// TIA Portal V19 export
DATA_BLOCK "DB_POS"   // DB51
{ S7_Optimized_Access := 'FALSE' }
AUTHOR : MS
// stored: AutoNumber false
   VAR RETAIN
      ANZAHL : Int := 58;   // Anzahl der Positionen
      Offset : Int := 50;   // * Beginn der Datenstruktur
      LENG : Int := 100;   // * Länge einer Position in Byte
      akt_POS : Int := 13;   // Position in Bearbeitung
      resW : Int := 0;
      resDW1 : DWord := 16#0000_0000;
      RESDW2 : DWord := 16#0000_0000;
      RESDW3 : DWord := 16#0000_0000;
      RESDW4 : DWord := 16#0000_0000;
      RESDW5 : DWord := 16#0000_0000;
      RESDW6 : DWord := 16#0000_0000;
      RESDW7 : DWord := 16#0000_0000;
      RESDW8 : DWord := 16#0000_0000;
      RESDW9 : DWord := 16#0000_0000;
      RESDW10 : DWord := 16#0000_0000;
      POS : Array[0..30] of Struct   // * Feldlänge anpassen
         Typ : Byte;   // Badtyp 0=Anlagenpos normal, 1-3=Be-Entladestand, 5=Speicher ,10=QT-Pos, 255 Dum
         SubTyp : Byte;   // Untertyp der Position 5=ExpoVorruf ignorieren bei 2xEinsetzen, 1=Sperre bei Alt
         Prio_Pos : Byte;   // Priorität des Bades (höchste Priorität==0
         SchiebePos : Byte;   // Position auf die FW geschoben wird, wenn er ohne Befehl hier steht
         Reihe : Byte;   // Reihe auf der sich die Position befindet
         FW_Nr : Byte;   // FW_Nr des FW, der über dieser Pos ist
         Optipos : Bool;   // WT wird in die Optimierungsrechnung einbezogen
         berechnet : Bool;   // WT wurde von der Optimierung berechnet
         Quelle : Bool;   // Position ist als Quelle reserviert
         Ziel : Bool;   // Position ist als Ziel reserviert
         FW_kommt : Bool;   // FW will dieses Bad überfahren
         FW_in_POS : Bool;   // Fahrwagen über Bad positioniert
         FW_Hebt : Bool;   // Fahrwagen hebt aus
         FW_Senkt : Bool;   // Fahrwagen setzt ein
         Sperre_in : Bool;   // Bad Einfahrsperre
         Sperre_FW : Bool;   // Bad Überfahrsperre
         Sperre_out : Bool;   // Bad Ausfahrsperre
         IN_OUT_nen : Bool;   // Einsetzen bzw. Ausheben nicht möglich, da Warenbewegung oder Deckel zu usw.
         lngsm_IN : Bool;   // langsames Einsetzen erforderlich-abhängig von immer_schnell
         lngsm_OUT : Bool;   // langsames Ausheben erforderlich-abhängig von immer_schnell
         immer_schnell : Bool;   // trockene Position (keine ATZ, schneller Hub erlaubt)
         QT_reserviert : Bool;   // Position ist durch QT reserviert
         KS_erlaubt : Bool;   // Pos darf mit KS befülltwerden
         LS_erlaubt : Bool;   // Pos darf mit LS befüllt werden
         GO_erlaubt : Bool;   // Pos darf mit GO befüllt werden
         Belegt_KS : Bool;   // Belegt mit KS
         Belegt_LS : Bool;   // Belegt mit LS
         Belegt_GO : Bool;   // Belegtmit GO
         Spr_Off : Bool;   // Oberhalb Z nicht spritzen
         Opt_Abgelehnt : Bool;   // Einfahrt durch Opti abgelehnt
         notFG_out : Bool;   // Position darf nicht geräumt werden (Merkersystem)
         notFG_in : Bool;   // Position darf nicht befüllt werden (Merkersystem)
         Anmeldung : Bool;   // bevorzugte Behandlung anmelden
         fPosfree : Bool;   // Folgeposition muß frei sein
         QT_Sperre : Bool;   // Position ist durch QT gesperrt FW darf Pos nicht bedienen
         Vorsperre : Bool;   // Einfahrsperre anmelden
         QT_FW_Ruf : Bool;   // QT wird auf dieser Position von einem FW benötigt
         QT_ext_Ruf : Bool;   // QT wird auf dieser Position von einem externen Gerät benötigt
         Bef_ende : Bool;   // in diesem Bad muß der Befehlsindex geschaltet werden
         DoppelTauch : Bool;   // Doppeltauchen angefordert
         ignor_Exp : Bool;   // Expozeit ignorieren (Transport)
         ignor_ESp : Bool;   // ignoriere Einfahrsperre (notFG_in)
         ignor_fPosFree : Bool;   // ignoriere fPosFree (z.B. für Freigabe Pos kurz vor Expoende)
         UebergabePos : Bool;   // Übergabe von Wts möglich
         Portable : Bool;   // Im Vorruf und transportierbar
         Checked : Bool;   // Position im ersten Check (FB9) geprüft
         Detailtyp : Byte;   // 0=egal, 11=KS. 12=LS, 20=GO (alleshex)
         BereichsTakte : Byte;   // 0=kein laden, ansonsten auf WTDB.DBB54
         Stand_Nr : Byte;   // Verweis auf Stand Nr
         Absetzhoehe : DInt;   // Absetzhöhe in Inkrementen
         LZ_Nr1 : Byte;   // Verweis auf Ladungszähler Nr1
         LZ_Nr2 : Byte;   // Verweis auf Ladungszähler Nr2
         ZG_1 : Byte;   // Reserve für weitere Verweise
         ZG_2 : Byte;   // Reserve für weitere Verweise
         IncPos : DInt;   // Position des Bades in der Anlage
         IncAbstand_vor : Int;   // min. Abstand zum Bad bei Überfahrsperre
         IncAbstand_rck : Int;   // min. Abstand zum Bad bei Überfahrsperre
         WT_Nr_lang : DInt;   // Warenträger-Nr.
         WT_Stangen_Nr : Byte;   // Stangen-Nr
         WT_DB : Byte;   // DB_Nr Warenstange
         next_WT : Byte;   // WT der sich für diese Pos anmeldet
         Prio : Bool;
         INA : Bool;
         INE : Bool;
         OUTA : Bool;
         OUTE : Bool;
         SpProg : Bool;
         ResAmTW : Bool;
         ResAmQT : Bool;
         Trommel : Bool;   // Kontrolle aktiviert
         Leer_WT : Bool;   // Leerwarenträger HFs aus
         Warnung : Bool;   // in Position wurde eine Warnmeldung ausgelöst
         Alarm : Bool;   // in Position wurde eine Alarmmeldung ausgelöst
         WT_neu : Bool;   // WT wurde vom LZ noch nicht berücksichtigt
         lngsm_Hub : Bool;   // langsam Heben als WT-Parameter
         B_Takte_Null : Bool;   // Bereichstakte sind Null
         enable_reload : Bool;   // laden der Altwerte innerhalb einer Gruppe erlaubt
         WT_Typ : Byte;   // Art des Warenträgers (z.Bsp. bei fester Zuordnung Ware-WT)
         WT_Befx : Int;   // WT Befehlsindex
         Soll_Takte : Int;   // VERWEILTAKTE
         Soll_Expozeit : DInt;   // Sollwert Expositionszeit
         ExpoToleranz : DInt;   // Toleranzwert für Expozeit
         KF_A : Real;   // Korrekturfaktor WT_Auslastung 0..100%-->0..1, Gesamtoberfläche
         KF_Expo : Real;   // Korrekturfaktor Expozeit
         Korr_Restzeit : DInt;   // korregierte Restzeit bis zur Abholung WT
         SonderPos_Offset : DInt;   // Offset für Positionierung außermittig (Höhenwechsel,Blende usw.)
         Restvorsperre : Int;   // Resttakte bis Vorsperre
         Resttakte : Int;   // Taktzähler
         Restzeit : DInt;   // verbleibende Expositionszeit
         Verweilzeit : DInt;   // Verweilzeit
         T_Vorruf : Int;   // Vorrufzeit lößt Vorruf n Sekunden vor Ablauf der Expozeit aus
         T_Pend : Int;   // Auspendelzeit 0..999s
         T_ATZ : Int;   // Abtropfzeit 0..999s
         T_Vorsperre : Int;   // Takte bis Vorsperre zu Sperre wird
         WaitTime : DInt;   // Zeit der Expounterbrechung
         Res_Real : Real;
         belegt : Bool;   // Bad belegt
         Bearbeitung : Bool;   // Badbehandlung läuft
         Vorruf : Bool;   // Bad FW-Vorruf
         fertig : Bool;   // Bad fertig
         AL_Expo : Bool;   // Expotoleranz um 30s überschritten
         Dkl_auf_Pos : Bool;
         Expo_Off : Bool;   // Expozeit unterbrochen (GR-Absenkung)
         yALEX : Bool;   // Alarm Expo auslösen
         US_on_Q : Bool;   // Ultraschall 7s einschalten, wenn Quelle
         AlExp : Bool;   // Alarm Expotoleranz war ein
         MD_Alex : Bool;   // Meldung Expoalarm wurde abgesetzt
         MD_res : Bool;   // Meldung Gleichrichterfehler
         MD_res_1 : Bool;   // Meldung Temperaturreglerfehler
         QT_in_Pos : Bool;   // QT in Position
         res27 : Bool;
         PendHub : Bool;   // Pendelhub aktiv
         Leerzeit : Int;   // Zeit welche Position nicht benutzt
      END_STRUCT;
      RESDW : DWord := 16#0000_0000;
   END_VAR
BEGIN
   POS[0].Typ := 16#00;
   POS[1].Typ := 16#03;
   POS[2..30].Typ := 16#00;
   POS[0..30].SubTyp := 16#00;
   POS[0..30].Prio_Pos := 16#05;
   POS[0..30].SchiebePos := 16#00;
   POS[0..30].Reihe := 16#01;
   POS[0..1].FW_Nr := 16#00;
   POS[2].FW_Nr := 16#01;
   POS[3..10].FW_Nr := 16#00;
   POS[11].FW_Nr := 16#02;
   POS[12..30].FW_Nr := 16#00;
   POS[0..30].Optipos := FALSE;
   POS[0..30].berechnet := FALSE;
   POS[0..30].Quelle := FALSE;
   POS[0..30].Ziel := FALSE;
   POS[0..30].FW_kommt := FALSE;
   POS[0..1].FW_in_POS := FALSE;
   POS[2].FW_in_POS := TRUE;
   POS[3..10].FW_in_POS := FALSE;
   POS[11].FW_in_POS := TRUE;
   POS[12..30].FW_in_POS := FALSE;
   POS[0..30].FW_Hebt := FALSE;
   POS[0..30].FW_Senkt := FALSE;
   POS[0..30].Sperre_in := FALSE;
   POS[0..30].Sperre_FW := FALSE;
   POS[0..30].Sperre_out := FALSE;
   POS[0..30].IN_OUT_nen := FALSE;
   POS[0..30].lngsm_IN := FALSE;
   POS[0..30].lngsm_OUT := FALSE;
   POS[0].immer_schnell := FALSE;
   POS[1..2].immer_schnell := TRUE;
   POS[3..27].immer_schnell := FALSE;
   POS[28].immer_schnell := TRUE;
   POS[29..30].immer_schnell := FALSE;
   POS[0..30].QT_reserviert := FALSE;
   POS[0..30].KS_erlaubt := FALSE;
   POS[0..30].LS_erlaubt := FALSE;
   POS[0..30].GO_erlaubt := FALSE;
   POS[0..30].Belegt_KS := FALSE;
   POS[0..30].Belegt_LS := FALSE;
   POS[0..30].Belegt_GO := FALSE;
   POS[0..30].Spr_Off := FALSE;
   POS[0..30].Opt_Abgelehnt := FALSE;
   POS[0].notFG_out := FALSE;
   POS[1].notFG_out := TRUE;
   POS[2..30].notFG_out := FALSE;
   POS[0].notFG_in := FALSE;
   POS[1].notFG_in := TRUE;
   POS[2..30].notFG_in := FALSE;
   POS[0..30].Anmeldung := FALSE;
   POS[0..30].fPosfree := FALSE;
   POS[0..30].QT_Sperre := FALSE;
   POS[0..30].Vorsperre := FALSE;
   POS[0..30].QT_FW_Ruf := FALSE;
   POS[0..30].QT_ext_Ruf := FALSE;
   POS[0..30].Bef_ende := TRUE;
   POS[0..30].DoppelTauch := FALSE;
   POS[0..30].ignor_Exp := FALSE;
   POS[0..30].ignor_ESp := FALSE;
   POS[0..30].ignor_fPosFree := FALSE;
   POS[0..30].UebergabePos := FALSE;
   POS[0..30].Portable := FALSE;
   POS[0..30].Checked := FALSE;
   POS[0..9].Detailtyp := 16#00;
   POS[10].Detailtyp := 16#16;
   POS[11..12].Detailtyp := 16#00;
   POS[13].Detailtyp := 16#15;
   POS[14].Detailtyp := 16#14;
   POS[15..16].Detailtyp := 16#00;
   POS[17].Detailtyp := 16#13;
   POS[18].Detailtyp := 16#00;
   POS[19].Detailtyp := 16#12;
   POS[20..21].Detailtyp := 16#00;
   POS[22].Detailtyp := 16#11;
   POS[23..30].Detailtyp := 16#00;
   POS[0..30].BereichsTakte := 16#00;
   POS[0].Stand_Nr := 16#00;
   POS[1].Stand_Nr := 16#01;
   POS[2..30].Stand_Nr := 16#00;
   POS[0..30].LZ_Nr1 := 16#00;
   POS[0..30].LZ_Nr2 := 16#00;
   POS[0..30].ZG_1 := 16#00;
   POS[0..30].ZG_2 := 16#00;
   POS[0].IncPos := 12000;
   POS[1].IncPos := 1000;
   POS[2].IncPos := 2000;
   POS[3].IncPos := 3000;
   POS[4].IncPos := 4000;
   POS[5].IncPos := 5000;
   POS[6].IncPos := 6000;
   POS[7].IncPos := 7000;
   POS[8].IncPos := 8000;
   POS[9].IncPos := 9000;
   POS[10].IncPos := 10000;
   POS[11].IncPos := 11000;
   POS[12].IncPos := 12000;
   POS[13].IncPos := 13000;
   POS[14].IncPos := 14000;
   POS[15].IncPos := 15000;
   POS[16].IncPos := 16000;
   POS[17].IncPos := 17000;
   POS[18].IncPos := 18000;
   POS[19].IncPos := 19000;
   POS[20].IncPos := 20000;
   POS[21].IncPos := 21000;
   POS[22].IncPos := 22000;
   POS[23].IncPos := 23000;
   POS[24].IncPos := 24000;
   POS[25].IncPos := 25000;
   POS[26].IncPos := 26000;
   POS[27].IncPos := 27000;
   POS[28].IncPos := 28000;
   POS[29].IncPos := 29000;
   POS[30].IncPos := 30000;
   POS[0].IncAbstand_vor := 0;
   POS[1].IncAbstand_vor := 600;
   POS[2..30].IncAbstand_vor := 0;
   POS[0].IncAbstand_rck := 0;
   POS[1].IncAbstand_rck := 300;
   POS[2..30].IncAbstand_rck := 0;
   POS[0..30].WT_Nr_lang := 0;
   POS[0..30].WT_Stangen_Nr := 16#00;
   POS[0..30].WT_DB := 16#00;
   POS[0..30].next_WT := 16#00;
   POS[0..30].Prio := FALSE;
   POS[0..30].INA := FALSE;
   POS[0..30].INE := FALSE;
   POS[0..30].OUTA := FALSE;
   POS[0..30].OUTE := FALSE;
   POS[0..30].SpProg := FALSE;
   POS[0..30].ResAmTW := FALSE;
   POS[0..30].ResAmQT := FALSE;
   POS[0..30].Trommel := FALSE;
   POS[0..30].Leer_WT := FALSE;
   POS[0..30].Warnung := FALSE;
   POS[0..30].Alarm := FALSE;
   POS[0..30].WT_neu := FALSE;
   POS[0..30].lngsm_Hub := FALSE;
   POS[0..30].B_Takte_Null := FALSE;
   POS[0..3].enable_reload := FALSE;
   POS[4..7].enable_reload := TRUE;
   POS[8..30].enable_reload := FALSE;
   POS[0..30].WT_Typ := 16#00;
   POS[0..30].WT_Befx := 0;
   POS[0..30].Soll_Takte := 0;
   POS[0].Soll_Expozeit := 5;
   POS[1].Soll_Expozeit := 0;
   POS[2].Soll_Expozeit := 360;
   POS[3].Soll_Expozeit := 60;
   POS[4..7].Soll_Expozeit := 1260;
   POS[8..9].Soll_Expozeit := 90;
   POS[10].Soll_Expozeit := 75;
   POS[11..12].Soll_Expozeit := 5;
   POS[13..14].Soll_Expozeit := 75;
   POS[15..16].Soll_Expozeit := 5;
   POS[17].Soll_Expozeit := 75;
   POS[18].Soll_Expozeit := 5;
   POS[19].Soll_Expozeit := 75;
   POS[20].Soll_Expozeit := 5;
   POS[21].Soll_Expozeit := 10;
   POS[22].Soll_Expozeit := 360;
   POS[23..27].Soll_Expozeit := 5;
   POS[28].Soll_Expozeit := 0;
   POS[29..30].Soll_Expozeit := 5;
   POS[0..30].ExpoToleranz := 600;
   POS[0..30].KF_A := 0.0;
   POS[0..30].KF_Expo := 0.0;
   POS[0..30].Korr_Restzeit := 0;
   POS[0..30].SonderPos_Offset := 0;
   POS[0..30].Restvorsperre := 0;
   POS[0..30].Resttakte := 0;
   POS[0..30].Restzeit := 0;
   POS[0..30].Verweilzeit := 0;
   POS[0..30].T_Vorruf := 30;
   POS[0..30].T_Pend := 1;
   POS[0].T_ATZ := 5;
   POS[1..2].T_ATZ := 0;
   POS[3..7].T_ATZ := 10;
   POS[8..9].T_ATZ := 5;
   POS[10].T_ATZ := 10;
   POS[11..12].T_ATZ := 5;
   POS[13..14].T_ATZ := 10;
   POS[15..16].T_ATZ := 5;
   POS[17].T_ATZ := 10;
   POS[18].T_ATZ := 5;
   POS[19].T_ATZ := 10;
   POS[20..21].T_ATZ := 5;
   POS[22].T_ATZ := 10;
   POS[23].T_ATZ := 5;
   POS[24..27].T_ATZ := 2;
   POS[28].T_ATZ := 0;
   POS[29].T_ATZ := 5;
   POS[30].T_ATZ := 2;
   POS[0..30].T_Vorsperre := 0;
   POS[0..30].WaitTime := 0;
   POS[0..30].Res_Real := 0.0;
   POS[0..30].belegt := FALSE;
   POS[0..30].Bearbeitung := FALSE;
   POS[0..30].Vorruf := FALSE;
   POS[0..30].fertig := FALSE;
   POS[0..30].AL_Expo := FALSE;
   POS[0..30].Dkl_auf_Pos := FALSE;
   POS[0..30].Expo_Off := FALSE;
   POS[0..30].yALEX := FALSE;
   POS[0..30].US_on_Q := FALSE;
   POS[0..30].AlExp := FALSE;
   POS[0..30].MD_Alex := FALSE;
   POS[0..30].MD_res := FALSE;
   POS[0..30].MD_res_1 := FALSE;
   POS[0..30].QT_in_Pos := FALSE;
   POS[0..30].res27 := FALSE;
   POS[0].PendHub := TRUE;
   POS[1..2].PendHub := FALSE;
   POS[3].PendHub := TRUE;
   POS[4..10].PendHub := FALSE;
   POS[11..12].PendHub := TRUE;
   POS[13..14].PendHub := FALSE;
   POS[15..16].PendHub := TRUE;
   POS[17].PendHub := FALSE;
   POS[18].PendHub := TRUE;
   POS[19].PendHub := FALSE;
   POS[20..21].PendHub := TRUE;
   POS[22].PendHub := FALSE;
   POS[23].PendHub := TRUE;
   POS[24..30].PendHub := FALSE;
   POS[0..30].Leerzeit := 32767;
END_DATA_BLOCK
